// TIA Portal project "greenhouse_plc_0.0.0" (V16)

(* hardware
DEVICE "S7-1200 station_1"  S7-1200 Station
   slot 0: "Telaio di montaggio_0"  S7-1200 Rack  Rack  V1.0
   slot 1: "PLC_1"  CPU 1211C DC/DC/DC  6ES7 211-1AE40-0XB0  V4.4
*)

// ===== PLC "PLC_1"  CPU 1211C DC/DC/DC =====

VAR_GLOBAL   // PLC tag table "Tabella delle variabili standard"
   "DI_cycle" AT %I0.0 : Bool;   // Start cycle
   "DI_stop" AT %I0.1 : Bool;   // Stop cycle
   "DI_start" AT %I0.2 : Bool;   // Start cycle
   "DI_emergency" AT %I0.3 : Bool;   // Emergency stop
   "DI_spare_1" AT %I0.4 : Bool;   // Spare 1
   "DI_spare_2" AT %I0.5 : Bool;   // Spare 2
   "DO_cycle" AT %Q0.0 : Bool;   // Cycle signal
   "DO_alarms" AT %Q0.1 : Bool;   // Alarms signal
   "System_Byte" AT %MB1 : Byte;
   "FirstScan" AT %M1.0 : Bool;
   "DiagStatusUpdate" AT %M1.1 : Bool;
   "AlwaysTRUE" AT %M1.2 : Bool;
   "AlwaysFALSE" AT %M1.3 : Bool;
   "Clock_Byte" AT %MB0 : Byte;
   "Clock_10Hz" AT %M0.0 : Bool;
   "Clock_5Hz" AT %M0.1 : Bool;
   "Clock_2.5Hz" AT %M0.2 : Bool;
   "Clock_2Hz" AT %M0.3 : Bool;
   "Clock_1.25Hz" AT %M0.4 : Bool;
   "Clock_1Hz" AT %M0.5 : Bool;
   "Clock_0.625Hz" AT %M0.6 : Bool;
   "Clock_0.5Hz" AT %M0.7 : Bool;
   "DO_light" AT %Q0.2 : Bool;   // Light
END_VAR

DATA_BLOCK "DB_Data"   // DB1
{ S7_Optimized_Access := 'FALSE' }
VERSION : 0.1
   VAR
      cycle_manual_mem : Bool;
      cycle_auto_mem : Bool;
      man_cycle : Bool;
      auto_cycle : Bool;
      alarm_presence : Bool;
      hmi_light_on : Bool;
      hmi_light_off : Bool;   // Luminosità
      hmi_start_cycle : Bool;
      hmi_light_mem : Bool;
      hmi_rain_mem : Bool;
      ss : Bool;
      ssss : Bool;
      Servo_Sx_Open : Bool;
      Servo_Sx_Close : Bool;
      Servo_Dx_Open : Bool;
      Servo_Dx_Close : Bool;
      "89" : Bool;
      "8" : Bool;
      "9" : Bool;
      cnt : Int;
      cnt_1 : Int;
      bo : Int;
      hmi_servo_dx_cmd_open : Int;
      hmi_servo_sx_cmd_open : Int;
      hmi_servo_dx_cmd_close : Int;
      hmi_servo_sx_cmd_close : Int;
      Servo_Sx_cmd : Int;
      Man_Aut_State : Int;
      Servo_State : Int;
      Automatic_Servo : Bool;
   END_VAR
BEGIN
END_DATA_BLOCK

DATA_BLOCK "DB_Arduino"   // DB2
{ S7_Optimized_Access := 'FALSE' }
VERSION : 0.1
   VAR
      Light : Int;
      Humidity : Int;
      Temperature : Int;
      Rain : Int;
      Servo_Dx_cmd : Int := 0;
      Servo_Sx_cmd : Int;
   END_VAR
BEGIN
END_DATA_BLOCK

DATA_BLOCK "DB_Alarms"   // DB4
{ S7_Optimized_Access := 'FALSE' }
VERSION : 0.1
   VAR
      alarm_0 : Bool;   // A000: emergency pressed
      alarm_1 : Bool;   // A001: min. light
      alarm_2 : Bool;   // A002: max. light
      alarm_3 : Bool;   // A003: min. humidity
      alarm_4 : Bool;   // A004: max. humidity
      alarm_5 : Bool;   // A005: min. temperature
      alarm_6 : Bool;   // A006: max. temperature
      alarm_7 : Bool;   // A007: min. rain
      alarm_8 : Bool;   // A008: max. rain
      alarm_9 : Bool;   // A009:
      alarm_10 : Bool;   // A010:
      alarm_11 : Bool;   // A011:
      alarm_12 : Bool;   // A012:
      alarm_13 : Bool;   // A013:
      alarm_14 : Bool;   // A014:
      alarm_15 : Bool;   // A015:
   END_VAR
BEGIN
END_DATA_BLOCK

DATA_BLOCK "DB_Settings"   // DB5
{ S7_Optimized_Access := 'FALSE' }
VERSION : 0.1
   VAR
      time_min_light : Time := T#10S;
      time_max_light : Time := T#10S;
      time_min_humidity : Time := T#10S;
      time_max_humidity : Time := T#10S;
      time_min_temperature : Time := T#10S;
      time_max_temperature : Time := T#10S;
      time_min_rain : Time := T#10S;
      time_max_rain : Time := T#10S;
      sp_min_light : Int := 55;
      sp_max_light : Int := 55;
      sp_min_humidity : Int := 40;
      sp_max_humidity : Int := 40;
      sp_min_temperature : Int := 25;
      sp_max_temperature : Int := 25;
      sp_min_rain : Int := 30;
      sp_max_rain : Int := 30;
      time_min_light_int : Int := 10;
      time_max_light_int : Int := 10;
      time_min_humidity_int : Int := 10;
      time_max_humidity_int : Int := 10;
      time_min_temperature_int : Int := 10;
      time_max_temperature_int : Int := 10;
      time_min_rain_int : Int := 10;
      time_max_rain_int : Int := 10;
   END_VAR
BEGIN
END_DATA_BLOCK

// folder: System blocks/Program resources

DATA_BLOCK "IEC_Counter_0_DB"   // DB3
{ S7_Optimized_Access := 'TRUE' }
AUTHOR : Simatic
FAMILY : IEC
NAME : CNTR
VERSION : 1.0
// stored: InstanceOfName IEC_COUNTER
"IEC_COUNTER"
BEGIN
END_DATA_BLOCK

DATA_BLOCK "IEC_Timer_0_DB"   // DB6
{ S7_Optimized_Access := 'TRUE' }
AUTHOR : Simatic
FAMILY : IEC
NAME : IEC_TMR
VERSION : 1.0
// stored: InstanceOfName IEC_TIMER
"IEC_TIMER"
BEGIN
END_DATA_BLOCK

DATA_BLOCK "IEC_Timer_1_DB"   // DB7
{ S7_Optimized_Access := 'TRUE' }
AUTHOR : Simatic
FAMILY : IEC
NAME : IEC_TMR
VERSION : 1.0
// stored: InstanceOfName IEC_TIMER
"IEC_TIMER"
BEGIN
END_DATA_BLOCK

DATA_BLOCK "IEC_Timer_2_DB"   // DB8
{ S7_Optimized_Access := 'TRUE' }
AUTHOR : Simatic
FAMILY : IEC
NAME : IEC_TMR
VERSION : 1.0
// stored: InstanceOfName IEC_TIMER
"IEC_TIMER"
BEGIN
END_DATA_BLOCK

DATA_BLOCK "IEC_Timer_3_DB"   // DB9
{ S7_Optimized_Access := 'TRUE' }
AUTHOR : Simatic
FAMILY : IEC
NAME : IEC_TMR
VERSION : 1.0
// stored: InstanceOfName IEC_TIMER
"IEC_TIMER"
BEGIN
END_DATA_BLOCK

DATA_BLOCK "IEC_Timer_4_DB"   // DB10
{ S7_Optimized_Access := 'TRUE' }
AUTHOR : Simatic
FAMILY : IEC
NAME : IEC_TMR
VERSION : 1.0
// stored: InstanceOfName IEC_TIMER
"IEC_TIMER"
BEGIN
END_DATA_BLOCK

DATA_BLOCK "IEC_Timer_5_DB"   // DB11
{ S7_Optimized_Access := 'TRUE' }
AUTHOR : Simatic
FAMILY : IEC
NAME : IEC_TMR
VERSION : 1.0
// stored: InstanceOfName IEC_TIMER
"IEC_TIMER"
BEGIN
END_DATA_BLOCK

DATA_BLOCK "IEC_Timer_6_DB"   // DB12
{ S7_Optimized_Access := 'TRUE' }
AUTHOR : Simatic
FAMILY : IEC
NAME : IEC_TMR
VERSION : 1.0
// stored: InstanceOfName IEC_TIMER
"IEC_TIMER"
BEGIN
END_DATA_BLOCK

DATA_BLOCK "IEC_Timer_7_DB"   // DB13
{ S7_Optimized_Access := 'TRUE' }
AUTHOR : Simatic
FAMILY : IEC
NAME : IEC_TMR
VERSION : 1.0
// stored: InstanceOfName IEC_TIMER
"IEC_TIMER"
BEGIN
END_DATA_BLOCK

// folder: (top level)

FUNCTION "0001_Cycle" : Void   // FC1, LAD
{ S7_Optimized_Access := 'TRUE' }
VERSION : 0.1
BEGIN

REGION Network 1: Start manual cycle
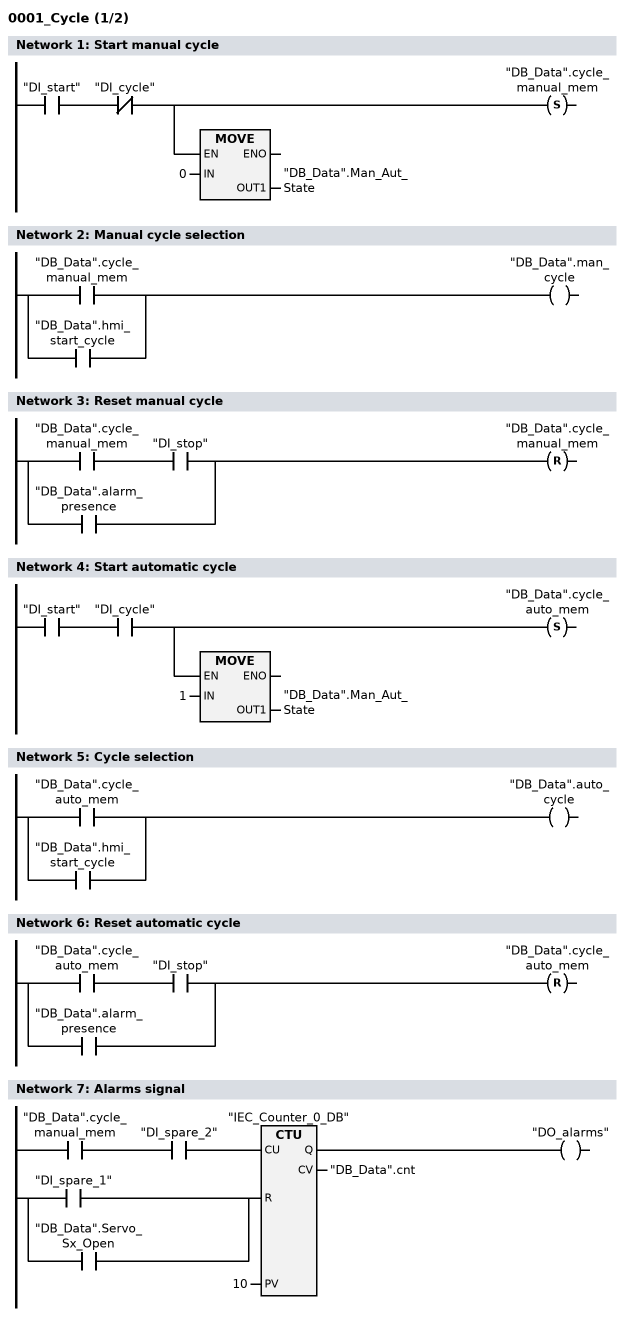
   RUNG wire#powerrail
      Contact( "DI_start" )
      I_Contact( "DI_cycle" )
      wire#w1
      S_Coil( "DB_Data".cycle_manual_mem )
   END_RUNG
   RUNG wire#w1
      Move(in := 0, out1 => "DB_Data".Man_Aut_State)
   END_RUNG
   // the same network as SCL:
   IF "DI_start" AND NOT "DI_cycle" THEN
       "DB_Data".cycle_manual_mem := TRUE;
       "DB_Data".Man_Aut_State := 0;
   END_IF;
END_REGION

REGION Network 2: Manual cycle selection
   RUNG wire#powerrail
      Contact( "DB_Data".cycle_manual_mem )
      wire#w1
      Coil( "DB_Data".man_cycle )
   END_RUNG
   RUNG wire#powerrail
      Contact( "DB_Data".hmi_start_cycle )
   END_RUNG wire#w1
   // the same network as SCL:
   "DB_Data".man_cycle := "DB_Data".cycle_manual_mem OR "DB_Data".hmi_start_cycle;
END_REGION

REGION Network 3: Reset manual cycle
   RUNG wire#powerrail
      Contact( "DB_Data".cycle_manual_mem )
      Contact( "DI_stop" )
      wire#w1
      R_Coil( "DB_Data".cycle_manual_mem )
   END_RUNG
   RUNG wire#powerrail
      Contact( "DB_Data".alarm_presence )
   END_RUNG wire#w1
   // the same network as SCL:
   IF ("DB_Data".cycle_manual_mem AND "DI_stop") OR "DB_Data".alarm_presence THEN
       "DB_Data".cycle_manual_mem := FALSE;
   END_IF;
END_REGION

REGION Network 4: Start automatic cycle
   RUNG wire#powerrail
      Contact( "DI_start" )
      Contact( "DI_cycle" )
      wire#w1
      S_Coil( "DB_Data".cycle_auto_mem )
   END_RUNG
   RUNG wire#w1
      Move(in := 1, out1 => "DB_Data".Man_Aut_State)
   END_RUNG
   // the same network as SCL:
   IF "DI_start" AND "DI_cycle" THEN
       "DB_Data".cycle_auto_mem := TRUE;
       "DB_Data".Man_Aut_State := 1;
   END_IF;
END_REGION

REGION Network 5: Cycle selection
   RUNG wire#powerrail
      Contact( "DB_Data".cycle_auto_mem )
      wire#w1
      Coil( "DB_Data".auto_cycle )
   END_RUNG
   RUNG wire#powerrail
      Contact( "DB_Data".hmi_start_cycle )
   END_RUNG wire#w1
   // the same network as SCL:
   "DB_Data".auto_cycle := "DB_Data".cycle_auto_mem OR "DB_Data".hmi_start_cycle;
END_REGION

REGION Network 6: Reset automatic cycle
   RUNG wire#powerrail
      Contact( "DB_Data".cycle_auto_mem )
      Contact( "DI_stop" )
      wire#w1
      R_Coil( "DB_Data".cycle_auto_mem )
   END_RUNG
   RUNG wire#powerrail
      Contact( "DB_Data".alarm_presence )
   END_RUNG wire#w1
   // the same network as SCL:
   IF ("DB_Data".cycle_auto_mem AND "DI_stop") OR "DB_Data".alarm_presence THEN
       "DB_Data".cycle_auto_mem := FALSE;
   END_IF;
END_REGION

REGION Network 7: Alarms signal
   "IEC_Counter_0_DB".CTU(CU := "DB_Data".cycle_manual_mem AND "DI_spare_2",
                          R := "DI_spare_1" OR "DB_Data".Servo_Sx_Open,
                          PV := 10,
                          CV => "DB_Data".cnt);
   "DO_alarms" := "IEC_Counter_0_DB".Q;
END_REGION

REGION Network 8: Manual light
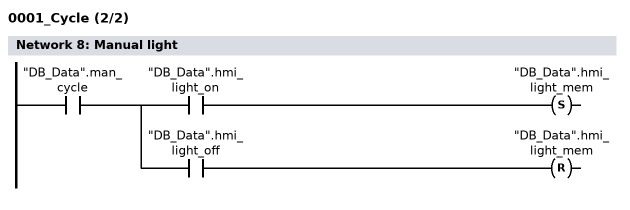
   RUNG wire#powerrail
      Contact( "DB_Data".man_cycle )
      wire#w1
      Contact( "DB_Data".hmi_light_on )
      S_Coil( "DB_Data".hmi_light_mem )
   END_RUNG
   RUNG wire#w1
      Contact( "DB_Data".hmi_light_off )
      R_Coil( "DB_Data".hmi_light_mem )
   END_RUNG
   // the same network as SCL:
   IF "DB_Data".man_cycle AND "DB_Data".hmi_light_on THEN "DB_Data".hmi_light_mem := TRUE; END_IF;
   IF "DB_Data".man_cycle AND "DB_Data".hmi_light_off THEN "DB_Data".hmi_light_mem := FALSE; END_IF;
END_REGION
END_FUNCTION

FUNCTION "0000_Alarms" : Void   // FC2, LAD
{ S7_Optimized_Access := 'TRUE' }
VERSION : 0.1
BEGIN

REGION Network 1: A000: emergency pressed
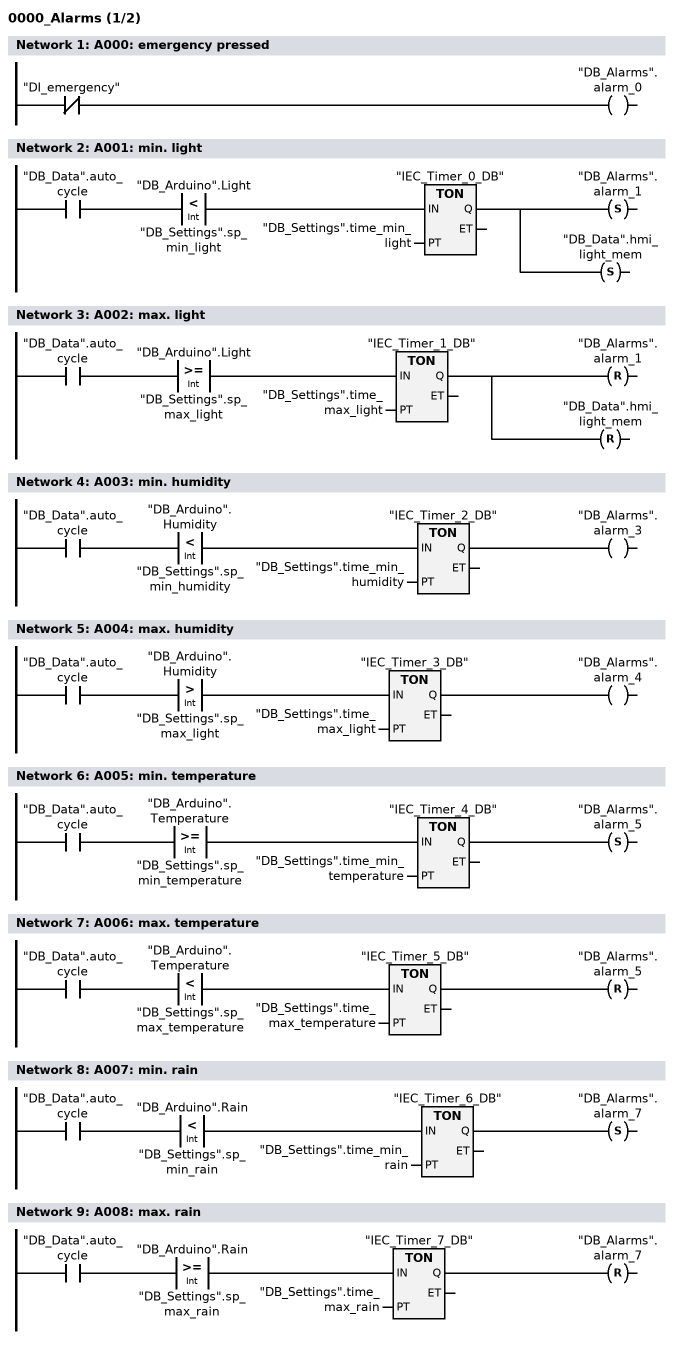
   RUNG wire#powerrail
      I_Contact( "DI_emergency" )
      Coil( "DB_Alarms".alarm_0 )
   END_RUNG
   // the same network as SCL:
   "DB_Alarms".alarm_0 := NOT "DI_emergency";
END_REGION

REGION Network 2: A001: min. light
   "IEC_Timer_0_DB".TON(IN := "DB_Data".auto_cycle AND ("DB_Arduino".Light < "DB_Settings".sp_min_light),
                        PT := "DB_Settings".time_min_light);
   IF "IEC_Timer_0_DB".Q THEN
       "DB_Alarms".alarm_1 := TRUE;
       "DB_Data".hmi_light_mem := TRUE;
   END_IF;
END_REGION

REGION Network 3: A002: max. light
   "IEC_Timer_1_DB".TON(IN := "DB_Data".auto_cycle AND ("DB_Arduino".Light >= "DB_Settings".sp_max_light),
                        PT := "DB_Settings".time_max_light);
   IF "IEC_Timer_1_DB".Q THEN
       "DB_Alarms".alarm_1 := FALSE;
       "DB_Data".hmi_light_mem := FALSE;
   END_IF;
END_REGION

REGION Network 4: A003: min. humidity
   "IEC_Timer_2_DB".TON(IN := "DB_Data".auto_cycle AND ("DB_Arduino".Humidity < "DB_Settings".sp_min_humidity),
                        PT := "DB_Settings".time_min_humidity);
   "DB_Alarms".alarm_3 := "IEC_Timer_2_DB".Q;
END_REGION

REGION Network 5: A004: max. humidity
   "IEC_Timer_3_DB".TON(IN := "DB_Data".auto_cycle AND ("DB_Arduino".Humidity > "DB_Settings".sp_max_light),
                        PT := "DB_Settings".time_max_light);
   "DB_Alarms".alarm_4 := "IEC_Timer_3_DB".Q;
END_REGION

REGION Network 6: A005: min. temperature
   "IEC_Timer_4_DB".TON(IN := "DB_Data".auto_cycle AND ("DB_Arduino".Temperature >= "DB_Settings".sp_min_temperature),
                        PT := "DB_Settings".time_min_temperature);
   IF "IEC_Timer_4_DB".Q THEN "DB_Alarms".alarm_5 := TRUE; END_IF;
END_REGION

REGION Network 7: A006: max. temperature
   "IEC_Timer_5_DB".TON(IN := "DB_Data".auto_cycle AND ("DB_Arduino".Temperature < "DB_Settings".sp_max_temperature),
                        PT := "DB_Settings".time_max_temperature);
   IF "IEC_Timer_5_DB".Q THEN "DB_Alarms".alarm_5 := FALSE; END_IF;
END_REGION

REGION Network 8: A007: min. rain
   "IEC_Timer_6_DB".TON(IN := "DB_Data".auto_cycle AND ("DB_Arduino".Rain < "DB_Settings".sp_min_rain),
                        PT := "DB_Settings".time_min_rain);
   IF "IEC_Timer_6_DB".Q THEN "DB_Alarms".alarm_7 := TRUE; END_IF;
END_REGION

REGION Network 9: A008: max. rain
   "IEC_Timer_7_DB".TON(IN := "DB_Data".auto_cycle AND ("DB_Arduino".Rain >= "DB_Settings".sp_max_rain),
                        PT := "DB_Settings".time_max_rain);
   IF "IEC_Timer_7_DB".Q THEN "DB_Alarms".alarm_7 := FALSE; END_IF;
END_REGION

REGION Network 10: Alarm presence
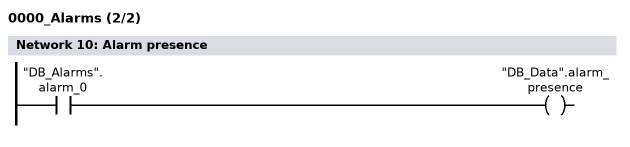
   RUNG wire#powerrail
      Contact( "DB_Alarms".alarm_0 )
      Coil( "DB_Data".alarm_presence )
   END_RUNG
   // the same network as SCL:
   "DB_Data".alarm_presence := "DB_Alarms".alarm_0;
END_REGION
END_FUNCTION

FUNCTION "0099_Command" : Void   // FC3, LAD
{ S7_Optimized_Access := 'TRUE' }
VERSION : 0.1
BEGIN

REGION Network 1: Cycle signaling
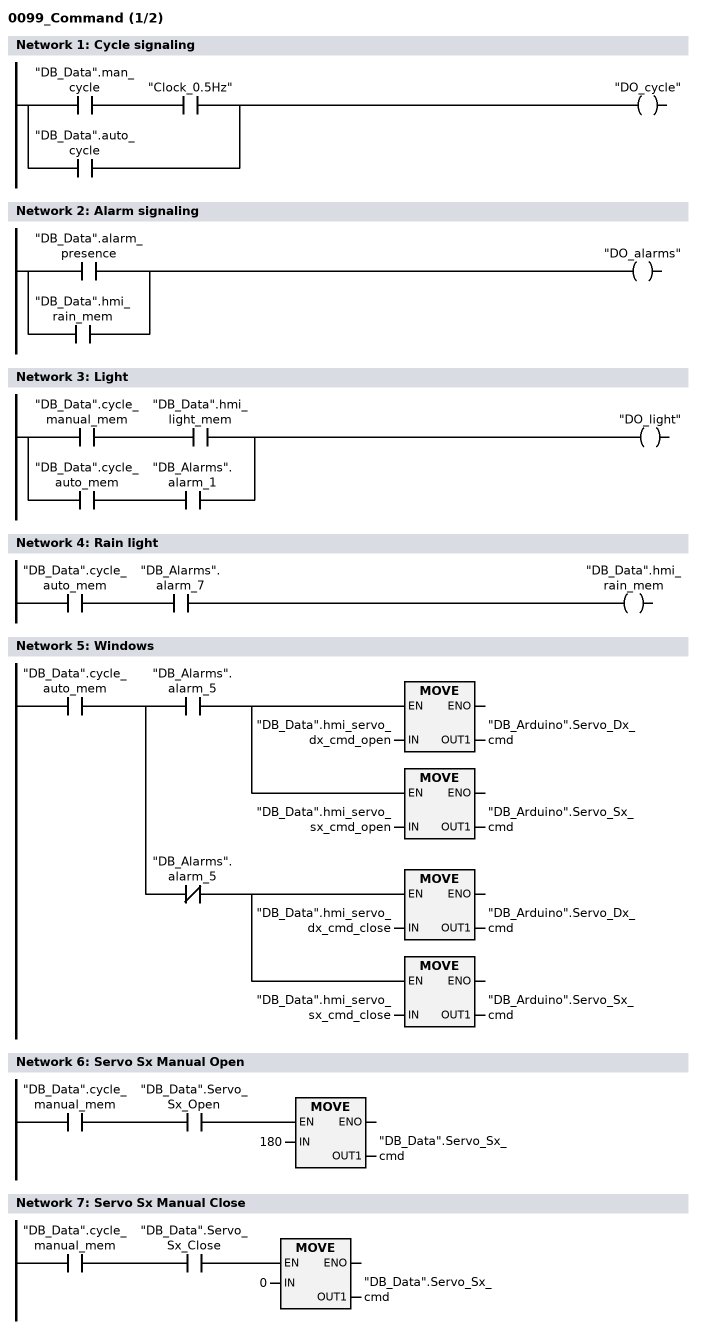
   RUNG wire#powerrail
      Contact( "DB_Data".man_cycle )
      Contact( "Clock_0.5Hz" )
      wire#w1
      Coil( "DO_cycle" )
   END_RUNG
   RUNG wire#powerrail
      Contact( "DB_Data".auto_cycle )
   END_RUNG wire#w1
   // the same network as SCL:
   "DO_cycle" := ("DB_Data".man_cycle AND "Clock_0.5Hz") OR "DB_Data".auto_cycle;
END_REGION

REGION Network 2: Alarm signaling
   RUNG wire#powerrail
      Contact( "DB_Data".alarm_presence )
      wire#w1
      Coil( "DO_alarms" )
   END_RUNG
   RUNG wire#powerrail
      Contact( "DB_Data".hmi_rain_mem )
   END_RUNG wire#w1
   // the same network as SCL:
   "DO_alarms" := "DB_Data".alarm_presence OR "DB_Data".hmi_rain_mem;
END_REGION

REGION Network 3: Light
   RUNG wire#powerrail
      Contact( "DB_Data".cycle_manual_mem )
      Contact( "DB_Data".hmi_light_mem )
      wire#w1
      Coil( "DO_light" )
   END_RUNG
   RUNG wire#powerrail
      Contact( "DB_Data".cycle_auto_mem )
      Contact( "DB_Alarms".alarm_1 )
   END_RUNG wire#w1
   // the same network as SCL:
   "DO_light" := ("DB_Data".cycle_manual_mem AND "DB_Data".hmi_light_mem) OR ("DB_Data".cycle_auto_mem AND "DB_Alarms".alarm_1);
END_REGION

REGION Network 4: Rain light
   RUNG wire#powerrail
      Contact( "DB_Data".cycle_auto_mem )
      Contact( "DB_Alarms".alarm_7 )
      Coil( "DB_Data".hmi_rain_mem )
   END_RUNG
   // the same network as SCL:
   "DB_Data".hmi_rain_mem := "DB_Data".cycle_auto_mem AND "DB_Alarms".alarm_7;
END_REGION

REGION Network 5: Windows
   RUNG wire#powerrail
      Contact( "DB_Data".cycle_auto_mem )
      wire#w1
      Contact( "DB_Alarms".alarm_5 )
      wire#w2
      Move(in := "DB_Data".hmi_servo_dx_cmd_open, out1 => "DB_Arduino".Servo_Dx_cmd)
   END_RUNG
   RUNG wire#w2
      Move(in := "DB_Data".hmi_servo_sx_cmd_open, out1 => "DB_Arduino".Servo_Sx_cmd)
   END_RUNG
   RUNG wire#w1
      I_Contact( "DB_Alarms".alarm_5 )
      wire#w3
      Move(in := "DB_Data".hmi_servo_dx_cmd_close, out1 => "DB_Arduino".Servo_Dx_cmd)
   END_RUNG
   RUNG wire#w3
      Move(in := "DB_Data".hmi_servo_sx_cmd_close, out1 => "DB_Arduino".Servo_Sx_cmd)
   END_RUNG
   // the same network as SCL:
   IF "DB_Data".cycle_auto_mem AND "DB_Alarms".alarm_5 THEN
       "DB_Arduino".Servo_Dx_cmd := "DB_Data".hmi_servo_dx_cmd_open;
       "DB_Arduino".Servo_Sx_cmd := "DB_Data".hmi_servo_sx_cmd_open;
   END_IF;
   IF "DB_Data".cycle_auto_mem AND NOT "DB_Alarms".alarm_5 THEN
       "DB_Arduino".Servo_Dx_cmd := "DB_Data".hmi_servo_dx_cmd_close;
       "DB_Arduino".Servo_Sx_cmd := "DB_Data".hmi_servo_sx_cmd_close;
   END_IF;
END_REGION

REGION Network 6: Servo Sx Manual Open
   RUNG wire#powerrail
      Contact( "DB_Data".cycle_manual_mem )
      Contact( "DB_Data".Servo_Sx_Open )
      Move(in := 180, out1 => "DB_Data".Servo_Sx_cmd)
   END_RUNG
   // the same network as SCL:
   IF "DB_Data".cycle_manual_mem AND "DB_Data".Servo_Sx_Open THEN "DB_Data".Servo_Sx_cmd := 180; END_IF;
END_REGION

REGION Network 7: Servo Sx Manual Close
   RUNG wire#powerrail
      Contact( "DB_Data".cycle_manual_mem )
      Contact( "DB_Data".Servo_Sx_Close )
      Move(in := 0, out1 => "DB_Data".Servo_Sx_cmd)
   END_RUNG
   // the same network as SCL:
   IF "DB_Data".cycle_manual_mem AND "DB_Data".Servo_Sx_Close THEN "DB_Data".Servo_Sx_cmd := 0; END_IF;
END_REGION

REGION Network 8: Servo Automatic Open
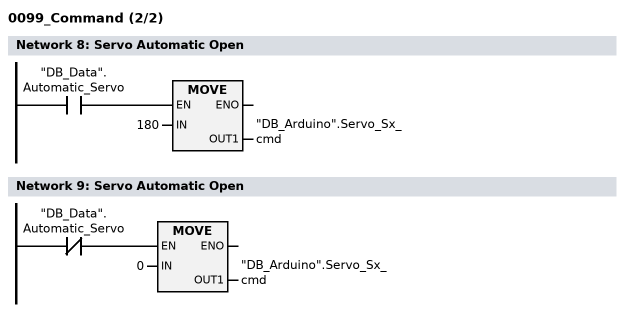
   RUNG wire#powerrail
      Contact( "DB_Data".Automatic_Servo )
      Move(in := 180, out1 => "DB_Arduino".Servo_Sx_cmd)
   END_RUNG
   // the same network as SCL:
   IF "DB_Data".Automatic_Servo THEN "DB_Arduino".Servo_Sx_cmd := 180; END_IF;
END_REGION

REGION Network 9: Servo Automatic Open
   RUNG wire#powerrail
      I_Contact( "DB_Data".Automatic_Servo )
      Move(in := 0, out1 => "DB_Arduino".Servo_Sx_cmd)
   END_RUNG
   // the same network as SCL:
   IF NOT "DB_Data".Automatic_Servo THEN "DB_Arduino".Servo_Sx_cmd := 0; END_IF;
END_REGION
END_FUNCTION

FUNCTION "0002_Settings" : Void   // FC4, LAD
{ S7_Optimized_Access := 'TRUE' }
VERSION : 0.1
BEGIN

REGION Network 1 (SCL)
   "DB_Settings".time_min_light := INT_TO_TIME("DB_Settings".time_min_light_int * 1000);
   "DB_Settings".time_max_light := INT_TO_TIME("DB_Settings".time_max_light_int * 1000);

   "DB_Settings".time_min_temperature := INT_TO_TIME("DB_Settings".time_min_temperature_int * 1000);
   "DB_Settings".time_max_temperature := INT_TO_TIME("DB_Settings".time_max_temperature_int * 1000);

   "DB_Settings".time_min_rain := INT_TO_TIME("DB_Settings".time_min_rain_int * 1000);
   "DB_Settings".time_max_rain := INT_TO_TIME("DB_Settings".time_max_rain_int * 1000);

   "DB_Settings".time_min_humidity := INT_TO_TIME("DB_Settings".time_min_humidity_int * 1000);
   "DB_Settings".time_max_humidity := INT_TO_TIME("DB_Settings".time_max_humidity_int * 1000);
END_REGION
END_FUNCTION

ORGANIZATION_BLOCK "Main"   // OB1, LAD, ProgramCycle
TITLE = "Main Program Sweep (Cycle)"
{ S7_Optimized_Access := 'TRUE' }
VERSION : 0.1
   VAR_INPUT
      Initial_Call : Bool;   // Initial call of this OB
      Remanence : Bool;   // =True, if remanent data are available
   END_VAR
BEGIN

REGION Network 1 (SCL): Main
   "0000_Alarms"();
   "0001_Cycle"();
   "0002_Settings"();
   "0099_Command"();
END_REGION
END_ORGANIZATION_BLOCK